// TIA Portal V17 export
// export: Created 2023-12-22T15:08:00.3717105Z, ExportSetting WithDefaults, DisplayName Totally Integrated Automation Portal, DisplayVersion V17, DisplayName TIA Portal Openness, DisplayVersion V17, DisplayName TIA Portal Version Control Interface, DisplayVersion V17, DisplayName STEP 7 Professional, DisplayVersion V17, DisplayName STEP 7 Safety, DisplayVersion V17, DisplayName WinCC Advanced, DisplayVersion V17
FUNCTION_BLOCK "Logick"   // FB1, LAD
{ S7_Optimized_Access := 'FALSE' }
VERSION : 0.1
// Mode - режим работы установки:
// 0 - поддержание давление
// 1 - поддержание уровня после насосной станции
// 2 - поддержание уровня до насосной станции
// stored: AutoNumber true, IsIECCheckEnabled false, SetENOAutomatically false, UDAEnableTagReadback false
   VAR_INPUT
      PE : Real;
      LE_Target : Real;
      LE_Source : Real := 3.0;
   END_VAR
   VAR DB_SPECIFIC
      Start : Bool;   // Общий запуск
      Dynamic : Bool;   // Динамический выбор кол-ва насосов
      Rotation : Bool;   // Ротация насосов
      Load : Bool;   // Ввод недостающего насоса
      Reload : Bool;   // Ввод резервного
      Deload : Bool;   // Вывод насоса при косяке
      PS_Add : Bool;   // +1 насос
      PS_Sub : Bool;   // -1 насос
      PE_Alarm : Bool;
      PE_Warning : Bool;
      LE_in_Alarm : Bool;
      LE_in_Warning : Bool;
      LE_out_Alarm : Bool;
      LE_out_Warning : Bool;
      Mode { S7_SetPoint := 'True'} : Int;   // Режим работы
      "Step" : Int;   // Глобальные этапы работы
      SP_Hz : Real;
      PS_REQ : Int;
      PS_cnt : Int;
      PE_SP { S7_SetPoint := 'True'} : Real;   // Уставка давления при работе
      PE_StartUp : Real;   // Уставка давления при разгоне
      PE_Work : Real;   // Уставка давления для PID-регулятора
      LE_Target_SP : Real;
      LE_Source_SP : Real;
      PID_Correction : Real;   // Поправка ПИД для заполнения по уровню
      SP_Low : Real := 40.0;   // Нижняя рабочая точка
      SP_High { S7_SetPoint := 'True'} : Real := 45.0;   // Верхняя рабочая точка
      SP_Min { S7_SetPoint := 'True'} : Real := 36.0;   // Точка открытия обратного клапана
      SP_PE_Alarm { S7_SetPoint := 'True'} : Real := 16.0;   // Аварийная точка давление - отключение насосной станции
      SP_PE_Warning { S7_SetPoint := 'True'} : Real := 14.5;   // Предупреждающее давление - блокировка разгона
      SP_LE_in_Warning { S7_SetPoint := 'True'} : Real := 2.0;
      SP_LE_in_Alarm { S7_SetPoint := 'True'} : Real := 1.0;
      SP_LE_out_Warning { S7_SetPoint := 'True'} : Real := 2.0;
      SP_LE_out_Alarm { S7_SetPoint := 'True'} : Real := 1.0;
      xPE : Real;   // Соотношение давления к уставке
      xPE_Min { S7_SetPoint := 'True'} : Real := 0.7;   // Минимальное соотношение
      Mode_5_REQ { S7_SetPoint := 'True'} : Int := 2;
      Mode_5_SP { S7_SetPoint := 'True'} : Real := 44.4;
      in_PE_LS { S7_SetPoint := 'True'} : Real := -0.4;   // Предупреждающе низкое давление всасывания
      in_PE_LLS { S7_SetPoint := 'True'} : Real := -0.8;   // Аварийно низкое давление всасывания
      Events : Word;
      Alarms : Word;
      pos : Array[0..15] of Bool;
   END_VAR
   VAR
      T_Delay_ADD { S7_SetPoint := 'True'} : "Time_M";   // Задержка добавления насоса
      T_Delay_SUB { S7_SetPoint := 'True'} : "Time_M";   // Задержка добавления насоса
      T_Rotation { S7_SetPoint := 'True'} : "Time_D";
      T_in_PE { S7_SetPoint := 'True'} : "Time_M";
   END_VAR
   VAR_TEMP
      ev : Bool;
   END_VAR
   // T_Delay_ADD.SP_S := 5;
   // T_Delay_SUB.SP_S := 5;
   VAR_TEMP   // added for the SCL form of the ladder/FBD networks
      _w1 : Bool;
      _w2 : Bool;
      _w3 : Bool;
      _w4 : Bool;
   END_VAR
BEGIN

REGION Network 1: Обработка управления насосной станцией
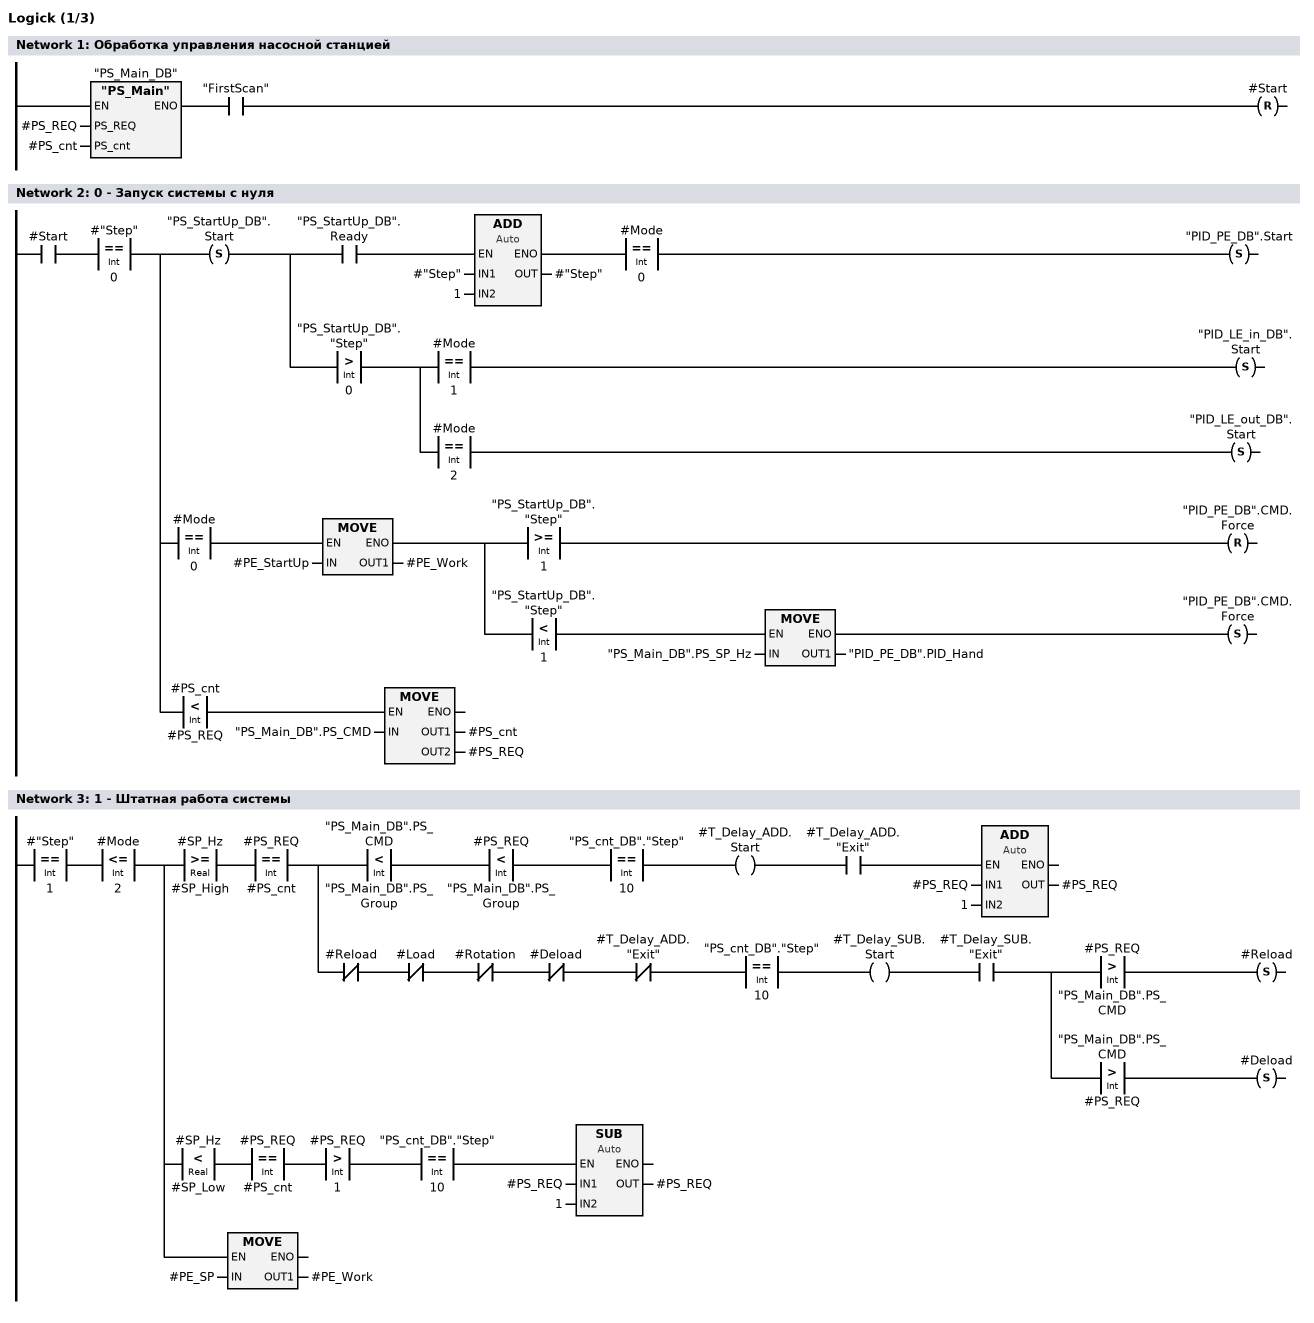
   RUNG wire#powerrail
      "PS_Main_DB"(PS_REQ := #PS_REQ, PS_cnt := #PS_cnt)
      Contact( "FirstScan" )
      R_Coil( #Start )
   END_RUNG
   // the same network as SCL:
   "PS_Main_DB"(PS_REQ := #PS_REQ, PS_cnt := #PS_cnt, ENO => #_w1);   // "PS_Main"
   IF #_w1 AND "FirstScan" THEN #Start := FALSE; END_IF;
END_REGION

REGION Network 2: 0 - Запуск системы с нуля
   RUNG wire#powerrail
      Contact( #Start )
      { S7_Templates := "SrcType := Int" } EQ_Contact(in1 := #"Step", in2 := 0)
      wire#w1
      S_Coil( "PS_StartUp_DB".Start )
      wire#w2
      Contact( "PS_StartUp_DB".Ready )
      Add(in1 := #"Step", in2 := 1, out => #"Step")
      { S7_Templates := "SrcType := Int" } EQ_Contact(in1 := #Mode, in2 := 0)
      S_Coil( "PID_PE_DB".Start )
   END_RUNG
   RUNG wire#w2
      { S7_Templates := "SrcType := Int" } GT_Contact(in1 := "PS_StartUp_DB"."Step", in2 := 0)
      wire#w3
      { S7_Templates := "SrcType := Int" } EQ_Contact(in1 := #Mode, in2 := 1)
      S_Coil( "PID_LE_in_DB".Start )
   END_RUNG
   RUNG wire#w3
      { S7_Templates := "SrcType := Int" } EQ_Contact(in1 := #Mode, in2 := 2)
      S_Coil( "PID_LE_out_DB".Start )
   END_RUNG
   RUNG wire#w1
      { S7_Templates := "SrcType := Int" } EQ_Contact(in1 := #Mode, in2 := 0)
      Move(in := #PE_StartUp, out1 => #PE_Work)
      wire#w4
      { S7_Templates := "SrcType := Int" } GE_Contact(in1 := "PS_StartUp_DB"."Step", in2 := 1)
      R_Coil( "PID_PE_DB".CMD.Force )
   END_RUNG
   RUNG wire#w4
      { S7_Templates := "SrcType := Int" } LT_Contact(in1 := "PS_StartUp_DB"."Step", in2 := 1)
      Move(in := "PS_Main_DB".PS_SP_Hz, out1 => "PID_PE_DB".PID_Hand)
      S_Coil( "PID_PE_DB".CMD.Force )
   END_RUNG
   RUNG wire#w1
      { S7_Templates := "SrcType := Int" } LT_Contact(in1 := #PS_cnt, in2 := #PS_REQ)
      Move(in := "PS_Main_DB".PS_CMD, out1 => #PS_cnt, out2 => #PS_REQ)
   END_RUNG
   // the same network as SCL:
   #_w1 := #Start AND (#"Step" = 0);
   IF #_w1 THEN "PS_StartUp_DB".Start := TRUE; END_IF;
   #_w2 := #_w1 AND "PS_StartUp_DB".Ready;
   IF #_w2 THEN #"Step" := #"Step" + 1; END_IF;
   IF #_w2 AND (#Mode = 0) THEN "PID_PE_DB".Start := TRUE; END_IF;
   #_w3 := #_w1 AND ("PS_StartUp_DB"."Step" > 0);
   IF #_w3 AND (#Mode = 1) THEN "PID_LE_in_DB".Start := TRUE; END_IF;
   IF #_w3 AND (#Mode = 2) THEN "PID_LE_out_DB".Start := TRUE; END_IF;
   #_w4 := #_w1 AND (#Mode = 0);
   IF #_w4 THEN #PE_Work := #PE_StartUp; END_IF;
   IF #_w4 AND ("PS_StartUp_DB"."Step" >= 1) THEN "PID_PE_DB".CMD.Force := FALSE; END_IF;
   IF #_w4 AND ("PS_StartUp_DB"."Step" < 1) THEN
       "PID_PE_DB".PID_Hand := "PS_Main_DB".PS_SP_Hz;
       "PID_PE_DB".CMD.Force := TRUE;
   END_IF;
   IF #_w1 AND (#PS_cnt < #PS_REQ) THEN
       #PS_cnt := "PS_Main_DB".PS_CMD;
       #PS_REQ := "PS_Main_DB".PS_CMD;
   END_IF;
END_REGION

REGION Network 3: 1 - Штатная работа системы
   RUNG wire#powerrail
      { S7_Templates := "SrcType := Int" } EQ_Contact(in1 := #"Step", in2 := 1)
      { S7_Templates := "SrcType := Int" } LE_Contact(in1 := #Mode, in2 := 2)
      wire#w1
      { S7_Templates := "SrcType := Real" } GE_Contact(in1 := #SP_Hz, in2 := #SP_High)
      { S7_Templates := "SrcType := Int" } EQ_Contact(in1 := #PS_REQ, in2 := #PS_cnt)
      wire#w2
      { S7_Templates := "SrcType := Int" } LT_Contact(in1 := "PS_Main_DB".PS_CMD, in2 := "PS_Main_DB".PS_Group)
      { S7_Templates := "SrcType := Int" } LT_Contact(in1 := #PS_REQ, in2 := "PS_Main_DB".PS_Group)
      { S7_Templates := "SrcType := Int" } EQ_Contact(in1 := "PS_cnt_DB"."Step", in2 := 10)
      Coil( #T_Delay_ADD.Start )
      Contact( #T_Delay_ADD."Exit" )
      Add(in1 := #PS_REQ, in2 := 1, out => #PS_REQ)
   END_RUNG
   RUNG wire#w2
      I_Contact( #Reload )
      I_Contact( #Load )
      I_Contact( #Rotation )
      I_Contact( #Deload )
      I_Contact( #T_Delay_ADD."Exit" )
      { S7_Templates := "SrcType := Int" } EQ_Contact(in1 := "PS_cnt_DB"."Step", in2 := 10)
      Coil( #T_Delay_SUB.Start )
      Contact( #T_Delay_SUB."Exit" )
      wire#w3
      { S7_Templates := "SrcType := Int" } GT_Contact(in1 := #PS_REQ, in2 := "PS_Main_DB".PS_CMD)
      S_Coil( #Reload )
   END_RUNG
   RUNG wire#w3
      { S7_Templates := "SrcType := Int" } GT_Contact(in1 := "PS_Main_DB".PS_CMD, in2 := #PS_REQ)
      S_Coil( #Deload )
   END_RUNG
   RUNG wire#w1
      { S7_Templates := "SrcType := Real" } LT_Contact(in1 := #SP_Hz, in2 := #SP_Low)
      { S7_Templates := "SrcType := Int" } EQ_Contact(in1 := #PS_REQ, in2 := #PS_cnt)
      { S7_Templates := "SrcType := Int" } GT_Contact(in1 := #PS_REQ, in2 := 1)
      { S7_Templates := "SrcType := Int" } EQ_Contact(in1 := "PS_cnt_DB"."Step", in2 := 10)
      Sub(in1 := #PS_REQ, in2 := 1, out => #PS_REQ)
   END_RUNG
   RUNG wire#w1
      Move(in := #PE_SP, out1 => #PE_Work)
   END_RUNG
   // the same network as SCL:
   #_w1 := (#"Step" = 1) AND (#Mode <= 2);
   #_w2 := #_w1 AND (#SP_Hz >= #SP_High) AND (#PS_REQ = #PS_cnt);
   #T_Delay_ADD.Start := #_w2 AND ("PS_Main_DB".PS_CMD < "PS_Main_DB".PS_Group) AND (#PS_REQ < "PS_Main_DB".PS_Group) AND ("PS_cnt_DB"."Step" = 10);
   IF #T_Delay_ADD.Start AND #T_Delay_ADD."Exit" THEN #PS_REQ := #PS_REQ + 1; END_IF;
   #T_Delay_SUB.Start := #_w2 AND NOT #Reload AND NOT #Load AND NOT #Rotation AND NOT #Deload AND NOT #T_Delay_ADD."Exit" AND ("PS_cnt_DB"."Step" = 10);
   #_w3 := #T_Delay_SUB.Start AND #T_Delay_SUB."Exit";
   IF #_w3 AND (#PS_REQ > "PS_Main_DB".PS_CMD) THEN #Reload := TRUE; END_IF;
   IF #_w3 AND ("PS_Main_DB".PS_CMD > #PS_REQ) THEN #Deload := TRUE; END_IF;
   IF #_w1 AND (#SP_Hz < #SP_Low) AND (#PS_REQ = #PS_cnt) AND (#PS_REQ > 1) AND ("PS_cnt_DB"."Step" = 10) THEN
       #PS_REQ := #PS_REQ - 1;
   END_IF;
   IF #_w1 THEN #PE_Work := #PE_SP; END_IF;
END_REGION

REGION Network 4: 1 - Штатная работа - макс производительность
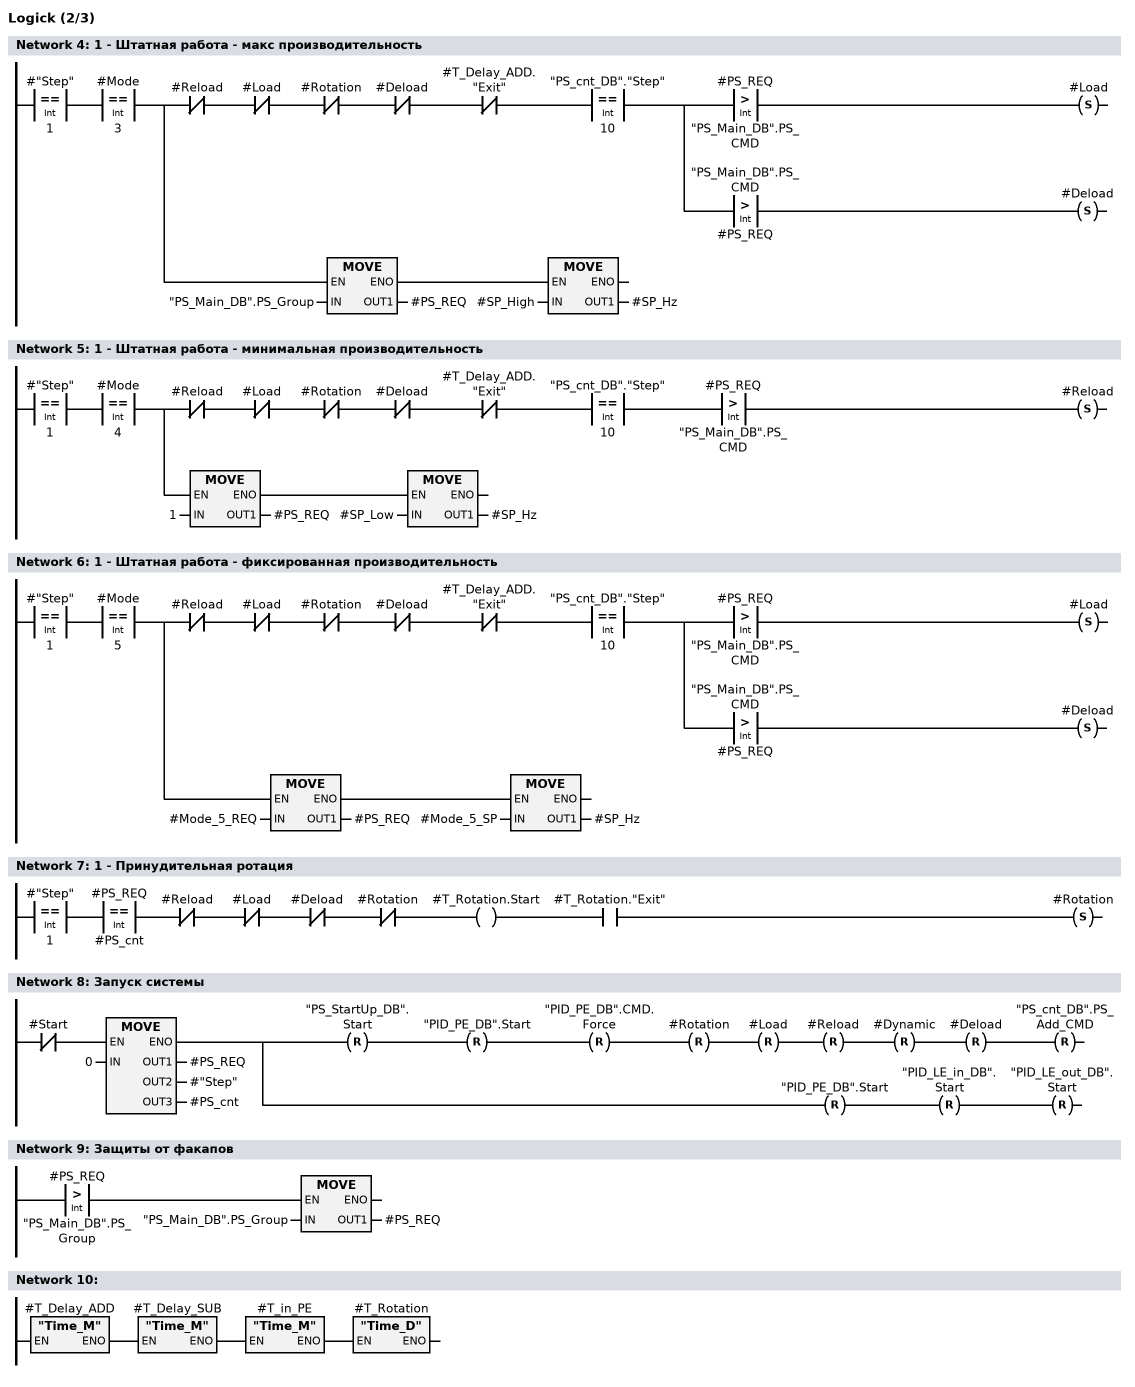
   RUNG wire#powerrail
      { S7_Templates := "SrcType := Int" } EQ_Contact(in1 := #"Step", in2 := 1)
      { S7_Templates := "SrcType := Int" } EQ_Contact(in1 := #Mode, in2 := 3)
      wire#w1
      I_Contact( #Reload )
      I_Contact( #Load )
      I_Contact( #Rotation )
      I_Contact( #Deload )
      I_Contact( #T_Delay_ADD."Exit" )
      { S7_Templates := "SrcType := Int" } EQ_Contact(in1 := "PS_cnt_DB"."Step", in2 := 10)
      wire#w2
      { S7_Templates := "SrcType := Int" } GT_Contact(in1 := #PS_REQ, in2 := "PS_Main_DB".PS_CMD)
      S_Coil( #Load )
   END_RUNG
   RUNG wire#w2
      { S7_Templates := "SrcType := Int" } GT_Contact(in1 := "PS_Main_DB".PS_CMD, in2 := #PS_REQ)
      S_Coil( #Deload )
   END_RUNG
   RUNG wire#w1
      Move(in := "PS_Main_DB".PS_Group, out1 => #PS_REQ)
      Move(in := #SP_High, out1 => #SP_Hz)
   END_RUNG
   // the same network as SCL:
   #_w1 := (#"Step" = 1) AND (#Mode = 3);
   #_w2 := #_w1 AND NOT #Reload AND NOT #Load AND NOT #Rotation AND NOT #Deload AND NOT #T_Delay_ADD."Exit" AND ("PS_cnt_DB"."Step" = 10);
   IF #_w2 AND (#PS_REQ > "PS_Main_DB".PS_CMD) THEN #Load := TRUE; END_IF;
   IF #_w2 AND ("PS_Main_DB".PS_CMD > #PS_REQ) THEN #Deload := TRUE; END_IF;
   IF #_w1 THEN
       #PS_REQ := "PS_Main_DB".PS_Group;
       #SP_Hz := #SP_High;
   END_IF;
END_REGION

REGION Network 5: 1 - Штатная работа - минимальная производительность
   RUNG wire#powerrail
      { S7_Templates := "SrcType := Int" } EQ_Contact(in1 := #"Step", in2 := 1)
      { S7_Templates := "SrcType := Int" } EQ_Contact(in1 := #Mode, in2 := 4)
      wire#w1
      I_Contact( #Reload )
      I_Contact( #Load )
      I_Contact( #Rotation )
      I_Contact( #Deload )
      I_Contact( #T_Delay_ADD."Exit" )
      { S7_Templates := "SrcType := Int" } EQ_Contact(in1 := "PS_cnt_DB"."Step", in2 := 10)
      { S7_Templates := "SrcType := Int" } GT_Contact(in1 := #PS_REQ, in2 := "PS_Main_DB".PS_CMD)
      S_Coil( #Reload )
   END_RUNG
   RUNG wire#w1
      Move(in := 1, out1 => #PS_REQ)
      Move(in := #SP_Low, out1 => #SP_Hz)
   END_RUNG
   // the same network as SCL:
   #_w1 := (#"Step" = 1) AND (#Mode = 4);
   IF #_w1 AND NOT #Reload AND NOT #Load AND NOT #Rotation AND NOT #Deload AND NOT #T_Delay_ADD."Exit" AND ("PS_cnt_DB"."Step" = 10) AND (#PS_REQ > "PS_Main_DB".PS_CMD) THEN
       #Reload := TRUE;
   END_IF;
   IF #_w1 THEN
       #PS_REQ := 1;
       #SP_Hz := #SP_Low;
   END_IF;
END_REGION

REGION Network 6: 1 - Штатная работа - фиксированная производительность
   RUNG wire#powerrail
      { S7_Templates := "SrcType := Int" } EQ_Contact(in1 := #"Step", in2 := 1)
      { S7_Templates := "SrcType := Int" } EQ_Contact(in1 := #Mode, in2 := 5)
      wire#w1
      I_Contact( #Reload )
      I_Contact( #Load )
      I_Contact( #Rotation )
      I_Contact( #Deload )
      I_Contact( #T_Delay_ADD."Exit" )
      { S7_Templates := "SrcType := Int" } EQ_Contact(in1 := "PS_cnt_DB"."Step", in2 := 10)
      wire#w2
      { S7_Templates := "SrcType := Int" } GT_Contact(in1 := #PS_REQ, in2 := "PS_Main_DB".PS_CMD)
      S_Coil( #Load )
   END_RUNG
   RUNG wire#w2
      { S7_Templates := "SrcType := Int" } GT_Contact(in1 := "PS_Main_DB".PS_CMD, in2 := #PS_REQ)
      S_Coil( #Deload )
   END_RUNG
   RUNG wire#w1
      Move(in := #Mode_5_REQ, out1 => #PS_REQ)
      Move(in := #Mode_5_SP, out1 => #SP_Hz)
   END_RUNG
   // the same network as SCL:
   #_w1 := (#"Step" = 1) AND (#Mode = 5);
   #_w2 := #_w1 AND NOT #Reload AND NOT #Load AND NOT #Rotation AND NOT #Deload AND NOT #T_Delay_ADD."Exit" AND ("PS_cnt_DB"."Step" = 10);
   IF #_w2 AND (#PS_REQ > "PS_Main_DB".PS_CMD) THEN #Load := TRUE; END_IF;
   IF #_w2 AND ("PS_Main_DB".PS_CMD > #PS_REQ) THEN #Deload := TRUE; END_IF;
   IF #_w1 THEN
       #PS_REQ := #Mode_5_REQ;
       #SP_Hz := #Mode_5_SP;
   END_IF;
END_REGION

REGION Network 7: 1 - Принудительная ротация
   RUNG wire#powerrail
      { S7_Templates := "SrcType := Int" } EQ_Contact(in1 := #"Step", in2 := 1)
      { S7_Templates := "SrcType := Int" } EQ_Contact(in1 := #PS_REQ, in2 := #PS_cnt)
      I_Contact( #Reload )
      I_Contact( #Load )
      I_Contact( #Deload )
      I_Contact( #Rotation )
      Coil( #T_Rotation.Start )
      Contact( #T_Rotation."Exit" )
      S_Coil( #Rotation )
   END_RUNG
   // the same network as SCL:
   #T_Rotation.Start := (#"Step" = 1) AND (#PS_REQ = #PS_cnt) AND NOT #Reload AND NOT #Load AND NOT #Deload AND NOT #Rotation;
   IF #T_Rotation.Start AND #T_Rotation."Exit" THEN #Rotation := TRUE; END_IF;
END_REGION

REGION Network 8: Запуск системы
   RUNG wire#powerrail
      I_Contact( #Start )
      Move(in := 0, out1 => #PS_REQ, out2 => #"Step", out3 => #PS_cnt)
      wire#w1
      R_Coil( "PS_StartUp_DB".Start )
      R_Coil( "PID_PE_DB".Start )
      R_Coil( "PID_PE_DB".CMD.Force )
      R_Coil( #Rotation )
      R_Coil( #Load )
      R_Coil( #Reload )
      R_Coil( #Dynamic )
      R_Coil( #Deload )
      R_Coil( "PS_cnt_DB".PS_Add_CMD )
   END_RUNG
   RUNG wire#w1
      R_Coil( "PID_PE_DB".Start )
      R_Coil( "PID_LE_in_DB".Start )
      R_Coil( "PID_LE_out_DB".Start )
   END_RUNG
   // the same network as SCL:
   IF NOT #Start THEN
       #PS_REQ := 0;
       #"Step" := 0;
       #PS_cnt := 0;
       "PS_StartUp_DB".Start := FALSE;
       "PID_PE_DB".Start := FALSE;
       "PID_PE_DB".CMD.Force := FALSE;
       #Rotation := FALSE;
       #Load := FALSE;
       #Reload := FALSE;
       #Dynamic := FALSE;
       #Deload := FALSE;
       "PS_cnt_DB".PS_Add_CMD := FALSE;
       "PID_PE_DB".Start := FALSE;
       "PID_LE_in_DB".Start := FALSE;
       "PID_LE_out_DB".Start := FALSE;
   END_IF;
END_REGION

REGION Network 9: Защиты от факапов
   RUNG wire#powerrail
      { S7_Templates := "SrcType := Int" } GT_Contact(in1 := #PS_REQ, in2 := "PS_Main_DB".PS_Group)
      Move(in := "PS_Main_DB".PS_Group, out1 => #PS_REQ)
   END_RUNG
   // the same network as SCL:
   IF #PS_REQ > "PS_Main_DB".PS_Group THEN #PS_REQ := "PS_Main_DB".PS_Group; END_IF;
END_REGION

REGION Network 10
   RUNG wire#powerrail
      #T_Delay_ADD()
      #T_Delay_SUB()
      #T_in_PE()
      #T_Rotation()
   END_RUNG
   // the same network as SCL:
   #T_Delay_ADD(ENO => #_w1);   // "Time_M"
   #T_Delay_SUB(EN := #_w1, ENO => #_w2);   // "Time_M"
   #T_in_PE(EN := #_w2, ENO => #_w3);   // "Time_M"
   IF #_w3 THEN
       #T_Rotation();   // "Time_D"
   END_IF;
END_REGION

REGION Network 11: Соотношение давления к уставке
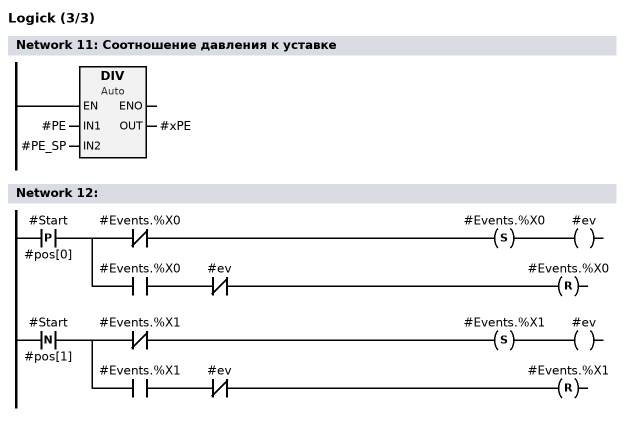
   RUNG wire#powerrail
      Div(in1 := #PE, in2 := #PE_SP, out => #xPE)
   END_RUNG
   // the same network as SCL:
   #xPE := #PE / #PE_SP;
END_REGION

REGION Network 12
   RUNG wire#powerrail
      P_Contact(operand := #Start, bit := #pos[0])
      wire#w1
      I_Contact( #Events.%X0 )
      S_Coil( #Events.%X0 )
      Coil( #ev )
   END_RUNG
   RUNG wire#w1
      Contact( #Events.%X0 )
      I_Contact( #ev )
      R_Coil( #Events.%X0 )
   END_RUNG
   RUNG wire#powerrail
      N_Contact(operand := #Start, bit := #pos[1])
      wire#w2
      I_Contact( #Events.%X1 )
      S_Coil( #Events.%X1 )
      Coil( #ev )
   END_RUNG
   RUNG wire#w2
      Contact( #Events.%X1 )
      I_Contact( #ev )
      R_Coil( #Events.%X1 )
   END_RUNG
   // the same network as SCL:
   #_w1 := #Start AND NOT #pos[0];   // rising edge of #Start
   #pos[0] := #Start;
   #_w2 := #_w1 AND NOT #Events.%X0;
   IF #_w2 THEN #Events.%X0 := TRUE; END_IF;
   #ev := #_w2;
   IF #_w1 AND #Events.%X0 AND NOT #ev THEN #Events.%X0 := FALSE; END_IF;
   #_w3 := NOT #Start AND #pos[1];   // falling edge of #Start
   #pos[1] := #Start;
   #_w4 := #_w3 AND NOT #Events.%X1;
   IF #_w4 THEN #Events.%X1 := TRUE; END_IF;
   #ev := #_w4;
   IF #_w3 AND #Events.%X1 AND NOT #ev THEN #Events.%X1 := FALSE; END_IF;
END_REGION
END_FUNCTION_BLOCK
